// TIA Portal V19 export
TYPE "LEXCHANGETRAY_typeConstraintWorkstation_signalTM_Monitor"
// stored: Access Published
   STRUCT
      simulationed : Bool;
      hookClawCylinderWorkPositionDetection2 : Bool;   // 钩爪气缸2工作位检测
      slideCylinderMedianPositionDetection1 : Bool;   // 滑台气缸中位检测1
      slideCylinderWorkPositionDetection1 : Bool;   // 滑台气缸工作位检测1
      motorConstraintPot2 : Bool;   // 拘束电机2正限
      motorConstraintNot2 : Bool;   // 拘束电机2负限
      motorConstraintPot1 : Bool;   // 拘束电机1正限
      motorConstraintOrg2 : Bool;   // 拘束电机2原点
      hookClawCylinderWorkPositionDetection1 : Bool;   // 钩爪气缸1工作位检测
      hookClawCylinderHomePositionDetection1 : Bool;   // 钩爪气缸1原位检测
      pressureGaugeSetValueDetection2_2 : Bool;   // 压力表2设定值检测2
      motorConstraintNot1 : Bool;   // 拘束电机1负限
      slideCylinderHomePositionDetection1 : Bool;   // 滑台气缸原位检测1
      motorConstraintOrg1 : Bool;   // 拘束电机1原点
      slideCylinderHomePositionDetection2 : Bool;   // 滑台气缸原位检测2
      pressureGaugeSetValueDetection1_2 : Bool;   // 压力表1设定值检测2
      pressureGaugeSetValueDetection2_1 : Bool;   // 压力表2设定值检测1
      slideCylinderWorkPositionDetection2 : Bool;   // 滑台气缸工作位检测2
      hookClawCylinderHomePositionDetection2 : Bool;   // 钩爪气缸2原位检测
      pressureGaugeSetValueDetection1_1 : Bool;   // 压力表1设定值检测1
      slideCylinderMedianPositionDetection2 : Bool;   // 滑台气缸中位检测2
   END_STRUCT;
END_TYPE
